TYPE tEncOutNCtrl1 :
STRUCT
	EnableLatchExternPositiveEdge		: BIT;
	SetCounter							: BIT;
	EnableLatchExternNegativeEdge		: BIT;
END_STRUCT
END_TYPE

(* stored: Version 1.1.0.1, ProductVersion 3.1.4024.10
   DUT tEncOutNCtrl1: Id {c31d0275-a13d-4b47-9358-f2566cfe8e9e} *)
